FUNCTION F_String_Builder : I_String_Builder
VAR_STAT
	fbString_Builder : FB_String_Builder;
END_VAR

fbString_Builder.Clear();
F_String_Builder := fbString_Builder;

END_FUNCTION

(* stored: Version 1.1.0.1, ProductVersion 3.1.4024.4
   POU F_String_Builder: Id {55e881ac-c530-44b9-b16a-c0ea1631cee2}, SpecialFunc None *)
